// Mitsubishi GX Works2 project: z20   PLC: Q02/Q02H

PROGRAM MAIN
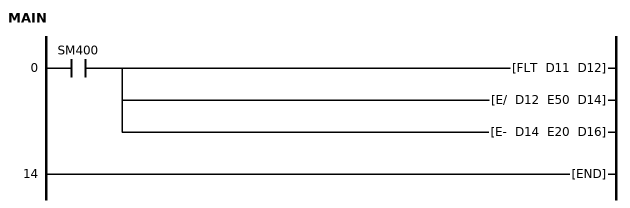
0     LD      SM400
      FLT     D11 D12
      E/      D12 E50 D14
      E-      D14 E20 D16
14    END
END_PROGRAM
